PROGRAM MAIN
VAR
END_VAR

MainASR();

END_PROGRAM

(* stored: Version 1.1.0.1
   POU MAIN: Id {7515210b-9d02-490f-8d89-bf94d83575cd}, SpecialFunc None *)
